{attribute 'GeneratedUsingTerminal: EK1100-0000-0018'}
{attribute addProperty BoxType "EK1100-0000-0018"}
{attribute addProperty Id "Beckhoff_EPP4xxxEK1122Beckhoff_EPP4xxxEK1122_696F89A1222"}
{attribute addProperty CRC "293499780"}
{attribute addProperty Size "222"}
TYPE Beckhoff_EPP4xxx_117E7384 EXTENDS EK1100_AB5A9467 :
STRUCT
	{attribute addProperty Name "Beckhoff_EPP4xxxEK1122"}
	Beckhoff_EPP4xxxEK1122 : Beckhoff_EPP4xxxEK1122_696F89A1;
END_STRUCT
END_TYPE

(* stored: Version 1.2.0.0, ProductVersion 3.1.4024.9
   DUT Beckhoff_EPP4xxx_117E7384: Id {58bd2a33-3344-4164-96a3-fc075d09aad4} *)
